PROGRAM PRG_DiagnosticPaddleMotors
VAR
    fbDPX_Motor : FB_MotionStage;
    fbDPY_Motor : FB_MotionStage;
    fbDPZ_Motor : FB_MotionStage;
END_VAR

fbDPX_Motor(stMotionStage:=PRG_Main.stDPXMotor);

fbDPY_Motor(stMotionStage:=PRG_Main.stDPYMotor);

fbDPZ_Motor(stMotionStage:=PRG_Main.stDPZMotor);

END_PROGRAM

(* stored: Version 1.1.0.1, ProductVersion 3.1.4024.6
   POU PRG_DiagnosticPaddleMotors: Id {698f952c-e0c1-49b9-9654-83f2078781a3}, SpecialFunc None *)
